(* IEC 61131-3 sources: thecodesysvibecoder/templates, 10 files *)

(* ---- FB_EtherCATMasterRestart.decl.st ---- *)
FUNCTION_BLOCK FB_EtherCATMasterRestart
VAR_INPUT
    xExecute : BOOL; // Rising edge starts a restart/reconfigure of the EtherCAT master connector.
    dwMasterModuleType : DWORD := DWORD#16#40; // IoStandard connector type CT_ETHERCAT_MASTER.
    dwMasterInstance : DWORD := 0; // EtherCAT master connector instance; normally 0 when there is one master.
END_VAR
VAR_OUTPUT
    xBusy : BOOL; // TRUE while IoMgrReconfigure is active.
    xDone : BOOL; // One-cycle pulse when the restart/reconfigure reports ASYNCSTATE_READY.
    xError : BOOL; // TRUE if the master connector cannot be found or reconfigure reports an error.
    xConnectorFound : BOOL; // TRUE when the EtherCAT master connector is found in the IoMgr connector list.
    dwMasterFlags : DWORD; // Raw IoConfigConnector.dwFlags of the master connector.
    udiConfigResult : UDINT; // Return code from IoMgrConfigGetConnectorList.
    udiReconfigureResult : UDINT; // Return code from IoMgrReconfigure.
    udiAsyncState : UDINT; // Async state: 0=pending, 1=active, 2=ready, 3=error, 4=timeout.
END_VAR
VAR
    pConnectorList : POINTER TO IoConfigConnector;
    pMasterConnector : POINTER TO IoConfigConnector;
    pActiveConnector : POINTER TO IoConfigConnector;
    diConnectorCount : DINT;
    xPrevExecute : BOOL; // Previous xExecute value for rising-edge detection.
    xStartRequest : BOOL; // Internal one-cycle request trigger.
    uiState : UINT; // 0=idle, 10=reconfigure active.
END_VAR

(* ---- FB_EtherCATOptionalSlaveManager.decl.st ---- *)
FUNCTION_BLOCK FB_EtherCATOptionalSlaveManager
VAR_INPUT
    xEnable : BOOL := TRUE; // FALSE leaves the EtherCAT master untouched by this FB.
    uiRequiredSlaves : UINT := 1; // Number of configured slaves that must be present; higher indexed slaves become optional.
    xApply : BOOL; // Rising edge reapplies optional flags and optionally restarts the master.
    xAutoApplyOnChange : BOOL := TRUE; // TRUE reapplies when uiRequiredSlaves changes.
    xRestartAfterApply : BOOL := TRUE; // TRUE pulses EtherCAT_Master.xRestart after optional flags are changed.
    xRestart : BOOL; // Manual rising edge pulses EtherCAT_Master.xRestart.
    xStepNonOperationalToOp : BOOL := TRUE; // TRUE tries INIT->PREOP->SAFEOP->OP for required slaves not yet operational.
    xStartConfigWithLessDevice : BOOL := TRUE; // Allows startup when optional configured slaves are not physically present.
    xAutoSetOperational : BOOL := TRUE; // Lets the master automatically retry optional/returning slaves.
    uiMaxSlavesToScan : UINT := 32; // Loop guard for the generated EtherCAT slave chain.
END_VAR
VAR_OUTPUT
    xDone : BOOL; // One-cycle pulse after optional flags were applied.
    xRestartPulse : BOOL; // TRUE for the cycle in which EtherCAT_Master.xRestart is pulsed.
    xConfigFinished : BOOL; // EtherCAT master reports that configuration download/startup is finished.
    xMasterError : BOOL; // EtherCAT master error output.
    xAnyNonOperational : BOOL; // TRUE when at least one scanned slave is not OP.
    uiConfiguredSlaves : UINT; // Number of slaves reached through EtherCAT_Master.FirstSlave/NextInstance.
    uiOptionalSlaves : UINT; // Number of scanned slaves above uiRequiredSlaves.
    uiOperationalSlaves : UINT; // Number of scanned slaves currently in OP.
    uiFirstNonOperationalIndex : UINT; // 1-based index of the first scanned slave not in OP; 0 when all are OP.
    eFirstNonOperationalState : ETC_SLAVE_STATE; // State of the first non-OP slave.
END_VAR
VAR
    pSlave : POINTER TO ETCSlave;
    uiIndex : UINT;
    xPrevApply : BOOL;
    xPrevRestart : BOOL;
    uiPrevRequiredSlaves : UINT := 65535;
    xApplyRequest : BOOL;
    xManualRestartRequest : BOOL;
    xDoRestart : BOOL;
    xOptional : BOOL;
END_VAR

(* ---- FB_IoConnectorRuntimeEnable.decl.st ---- *)
FUNCTION_BLOCK FB_IoConnectorRuntimeEnable
VAR_INPUT
    xEnable : BOOL := TRUE; // Requested runtime state for the selected I/O connector.
    xApply : BOOL; // Optional rising edge that applies the current request immediately.
    xAutoApplyOnChange : BOOL := TRUE; // TRUE applies automatically whenever xEnable changes.
    dwModuleType : DWORD := DWORD#16#41; // IoStandard module type; 16#41 is an EtherCAT slave connector in this project.
    dwInstance : DWORD := 1; // Connector instance: normally 0=first EtherCAT slave, 1=second, 2=third, etc.
    xUseCachedConnector : BOOL := TRUE; // Allows re-enable when a disabled connector is no longer returned by the active list.
END_VAR
VAR_OUTPUT
    xBusy : BOOL; // TRUE while IoMgrReconfigure is active.
    xDone : BOOL; // One-cycle pulse when reconfiguration reports ASYNCSTATE_READY.
    xError : BOOL; // TRUE if no usable connector exists or reconfiguration reports an error.
    xConnectorFound : BOOL; // TRUE when the connector is found in the current IoMgr connector list.
    xTargetAvailable : BOOL; // TRUE when either the current connector or a cached connector can be used.
    xUsingCachedConnector : BOOL; // TRUE when the FB is using the cached connector pointer for this cycle.
    xCurrentEnable : BOOL; // Current CF_ENABLE + CF_DEVICE_ENABLED flag state on the target connector.
    dwCurrentFlags : DWORD; // Raw IoConfigConnector.dwFlags of the target connector.
    udiConfigResult : UDINT; // Return code from IoMgrConfigGetConnectorList.
    udiReconfigureResult : UDINT; // Return code from IoMgrReconfigure.
    udiAsyncState : UDINT; // Async state: 0=pending, 1=active, 2=ready, 3=error, 4=timeout.
END_VAR
VAR
    pConnectorList : POINTER TO IoConfigConnector;
    pFoundConnector : POINTER TO IoConfigConnector;
    pTargetConnector : POINTER TO IoConfigConnector;
    pCachedConnector : POINTER TO IoConfigConnector;
    pActiveConnector : POINTER TO IoConfigConnector;
    diConnectorCount : DINT;
    xHaveCachedConnector : BOOL; // TRUE after the target connector was found at least once.
    xPrevApply : BOOL; // Previous xApply value for rising-edge detection.
    xPrevEnable : BOOL := TRUE; // Previous xEnable value for automatic change detection.
    xStartRequest : BOOL; // Internal one-cycle request trigger.
    uiState : UINT; // 0=idle, 10=reconfigure active.
END_VAR

(* ---- FB_MD5Hash.decl.st ---- *)
FUNCTION_BLOCK FB_MD5Hash
VAR_INPUT
    xExecute : BOOL; // Rising edge starts a new MD5 calculation.
    pData : POINTER TO BYTE; // Start address of the data to hash, normally ADR(stYourData).
    udiSize : UDINT; // Number of bytes to hash, normally SIZEOF(stYourData).
    abyExpectedDigest : ARRAY [0..15] OF BYTE; // Optional MD5 digest received from the other controller.
    xCompareExpected : BOOL := TRUE; // When TRUE, xMatch is updated when the local digest is done.
END_VAR
VAR_OUTPUT
    xDone : BOOL; // TRUE after a successful calculation; reset by the next xExecute rising edge.
    xBusy : BOOL; // TRUE while the CAA Memory MD5 block is calculating.
    xError : BOOL; // TRUE if a request is invalid, for example null pointer or zero byte length.
    xMatch : BOOL; // TRUE when the calculated digest equals abyExpectedDigest.
    abyDigest : ARRAY [0..15] OF BYTE; // Calculated 16-byte MD5 digest.
END_VAR
VAR
    fbMd5 : MEM.MD5; // CAA Memory MD5 function block.
    xExecuteOld : BOOL; // Previous xExecute state for rising-edge detection.
    xStart : BOOL; // One-cycle start pulse forwarded to MEM.MD5.
    i : INT; // Digest byte loop index.
END_VAR

(* ---- FB_S10eRuntimeEnable.decl.st ---- *)
FUNCTION_BLOCK FB_S10eRuntimeEnable
VAR_INPUT
    xEnableS10e1 : BOOL := TRUE; // Requested runtime state for the selected S10e EtherCAT slave.
    xApply : BOOL; // Optional rising edge that applies the current request immediately.
    xAutoApplyOnChange : BOOL := TRUE; // TRUE applies automatically whenever xEnableS10e1 changes.
    dwSlaveInstance : DWORD := 1; // Connector instance: normally 0=first S10e, 1=second, 2=third, etc.
    dwModuleType : DWORD := DWORD#16#41; // IoStandard module type; 16#41 is an EtherCAT slave connector in this project.
    xUseCachedConnector : BOOL := TRUE; // Allows re-enable when a disabled connector is no longer returned by the active list.
END_VAR
VAR_OUTPUT
    xBusy : BOOL; // TRUE while IoMgrReconfigure is active.
    xDone : BOOL; // One-cycle pulse when reconfiguration reports ASYNCSTATE_READY.
    xError : BOOL; // TRUE if no usable connector exists or reconfiguration reports an error.
    xConnectorFound : BOOL; // TRUE when the connector is found in the current IoMgr connector list.
    xTargetAvailable : BOOL; // TRUE when either the current connector or a cached connector can be used.
    xUsingCachedConnector : BOOL; // TRUE when the FB is using the cached connector pointer for this cycle.
    xCurrentEnable : BOOL; // Current CF_ENABLE + CF_DEVICE_ENABLED flag state on the target connector.
    dwCurrentFlags : DWORD; // Raw IoConfigConnector.dwFlags of the target connector.
    udiConfigResult : UDINT; // Return code from IoMgrConfigGetConnectorList.
    udiReconfigureResult : UDINT; // Return code from IoMgrReconfigure.
    udiAsyncState : UDINT; // Async state: 0=pending, 1=active, 2=ready, 3=error, 4=timeout.
END_VAR
VAR
    pConnectorList : POINTER TO IoConfigConnector;
    pFoundConnector : POINTER TO IoConfigConnector;
    pTargetConnector : POINTER TO IoConfigConnector;
    pCachedConnector : POINTER TO IoConfigConnector;
    pActiveConnector : POINTER TO IoConfigConnector;
    diConnectorCount : DINT;
    xHaveCachedConnector : BOOL; // TRUE after the target connector was found at least once.
    xPrevApply : BOOL; // Previous xApply value for rising-edge detection.
    xPrevEnableS10e1 : BOOL := TRUE; // Previous enable request for auto-apply change detection.
    xStartRequest : BOOL; // Internal one-cycle request trigger.
    uiState : UINT; // 0=idle, 10=reconfigure active.
END_VAR

(* ---- FB_EtherCATMasterRestart.impl.st ---- *)
// Restart/reconfigure the complete EtherCAT master connector.
// IoMgrReconfigure performs an asynchronous disable/enable/update-mapping
// sequence for the connector, which is the closest runtime "master restart"
// available through IoStandard.
xDone := FALSE;
xStartRequest := FALSE;

IF xExecute AND NOT xPrevExecute THEN
    xStartRequest := TRUE;
END_IF
xPrevExecute := xExecute;

udiConfigResult := IoMgrConfigGetConnectorList(
    ppConnectorList := ADR(pConnectorList),
    pnCount := ADR(diConnectorCount));

pMasterConnector := IoMgrConfigGetConnector(
    pConnectorList := pConnectorList,
    pnCount := ADR(diConnectorCount),
    dwModuleType := dwMasterModuleType,
    dwInstance := dwMasterInstance);

IF pMasterConnector <> 0 THEN
    xConnectorFound := TRUE;
    dwMasterFlags := pMasterConnector^.dwFlags;
ELSE
    xConnectorFound := FALSE;
    dwMasterFlags := DWORD#0;
END_IF

CASE uiState OF
    0:
        xBusy := FALSE;
        udiReconfigureResult := UDINT#0;

        IF xStartRequest THEN
            IF (udiConfigResult <> UDINT#0) OR NOT xConnectorFound THEN
                xError := TRUE;
            ELSE
                xError := FALSE;
                udiAsyncState := UDINT#16#FFFFFFFF;
                pActiveConnector := pMasterConnector;
                uiState := 10;
            END_IF
        END_IF

    10:
        xBusy := TRUE;
        IF pActiveConnector = 0 THEN
            xBusy := FALSE;
            xError := TRUE;
            uiState := 0;
        ELSE
            udiReconfigureResult := IoMgrReconfigure(
                pConnector := pActiveConnector,
                pudiState := ADR(udiAsyncState));

            dwMasterFlags := pActiveConnector^.dwFlags;

            IF udiReconfigureResult <> UDINT#0 THEN
                xBusy := FALSE;
                xError := TRUE;
                uiState := 0;
            ELSIF udiAsyncState = UDINT#2 THEN
                xBusy := FALSE;
                xDone := TRUE;
                xError := FALSE;
                uiState := 0;
            ELSIF (udiAsyncState = UDINT#3) OR (udiAsyncState = UDINT#4) THEN
                xBusy := FALSE;
                xError := TRUE;
                uiState := 0;
            END_IF
        END_IF

ELSE
    xBusy := FALSE;
    xError := TRUE;
    uiState := 0;
END_CASE

(* ---- FB_EtherCATOptionalSlaveManager.impl.st ---- *)
// Use the EtherCAT driver's optional-slave support instead of disabling
// IoStandard connectors. Disabled connectors can disappear from the runtime
// configuration and may not come back until a controller warm restart.
xDone := FALSE;
xRestartPulse := FALSE;
xApplyRequest := FALSE;
xManualRestartRequest := FALSE;

IF NOT xEnable THEN
    RETURN;
END_IF

IF xApply AND NOT xPrevApply THEN
    xApplyRequest := TRUE;
END_IF

IF xRestart AND NOT xPrevRestart THEN
    xManualRestartRequest := TRUE;
END_IF

IF xAutoApplyOnChange AND (uiRequiredSlaves <> uiPrevRequiredSlaves) THEN
    xApplyRequest := TRUE;
END_IF

xPrevApply := xApply;
xPrevRestart := xRestart;

// These properties must be set before or while the master starts.
EtherCAT_Master.StartConfigWithLessDevice := xStartConfigWithLessDevice;
EtherCAT_Master.AutoSetOperational := xAutoSetOperational;

IF xApplyRequest THEN
    pSlave := EtherCAT_Master.FirstSlave;
    uiIndex := 1;

    WHILE (pSlave <> 0) AND (uiIndex <= uiMaxSlavesToScan) DO
        // Slaves after uiRequiredSlaves remain in the configuration but are optional.
        xOptional := uiIndex > uiRequiredSlaves;
        pSlave^.SetOptional(xOptional);

        pSlave := pSlave^.NextInstance;
        uiIndex := uiIndex + 1;
    END_WHILE

    uiPrevRequiredSlaves := uiRequiredSlaves;
    xDone := TRUE;
END_IF

xDoRestart := xManualRestartRequest OR (xApplyRequest AND xRestartAfterApply);
EtherCAT_Master.xRestart := xDoRestart;
xRestartPulse := xDoRestart;

// The generated master instance must be called for xRestart and status updates.
EtherCAT_Master();

xConfigFinished := EtherCAT_Master.xConfigFinished;
xMasterError := EtherCAT_Master.xError;

uiConfiguredSlaves := 0;
uiOptionalSlaves := 0;
uiOperationalSlaves := 0;
uiFirstNonOperationalIndex := 0;
xAnyNonOperational := FALSE;
eFirstNonOperationalState := ETC_SLAVE_STATE.ETC_SLAVE_BOOT;

pSlave := EtherCAT_Master.FirstSlave;
uiIndex := 1;

WHILE (pSlave <> 0) AND (uiIndex <= uiMaxSlavesToScan) DO
    pSlave^();
    uiConfiguredSlaves := uiConfiguredSlaves + 1;

    xOptional := uiIndex > uiRequiredSlaves;
    IF xOptional THEN
        uiOptionalSlaves := uiOptionalSlaves + 1;
    END_IF

    IF pSlave^.wState = ETC_SLAVE_STATE.ETC_SLAVE_OPERATIONAL THEN
        uiOperationalSlaves := uiOperationalSlaves + 1;
    ELSE
        xAnyNonOperational := TRUE;
        IF uiFirstNonOperationalIndex = 0 THEN
            uiFirstNonOperationalIndex := uiIndex;
            eFirstNonOperationalState := pSlave^.wState;
        END_IF

        // Required slaves are actively stepped toward OP. Optional slaves are
        // handled by AutoSetOperational when they are connected again.
        IF xStepNonOperationalToOp AND xConfigFinished AND NOT xOptional THEN
            CASE pSlave^.wState OF
                ETC_SLAVE_STATE.ETC_SLAVE_INIT:
                    pSlave^.SetOpMode(ETC_SLAVE_STATE.ETC_SLAVE_PREOPERATIONAL);
                ETC_SLAVE_STATE.ETC_SLAVE_PREOPERATIONAL:
                    pSlave^.SetOpMode(ETC_SLAVE_STATE.ETC_SLAVE_SAVEOPERATIONAL);
                ETC_SLAVE_STATE.ETC_SLAVE_SAVEOPERATIONAL:
                    pSlave^.SetOpMode(ETC_SLAVE_STATE.ETC_SLAVE_OPERATIONAL);
            END_CASE
        END_IF
    END_IF

    pSlave := pSlave^.NextInstance;
    uiIndex := uiIndex + 1;
END_WHILE

(* ---- FB_IoConnectorRuntimeEnable.impl.st ---- *)
// Generic low-level runtime enable/disable for an IoStandard connector.
// For S10e EtherCAT slaves in this project, use dwModuleType 16#41 and select
// the unit by dwInstance. The CODESYS object name is not needed at runtime.
xDone := FALSE;
xStartRequest := FALSE;
xUsingCachedConnector := FALSE;

IF xApply AND NOT xPrevApply THEN
    xStartRequest := TRUE;
END_IF

IF xAutoApplyOnChange AND (xEnable <> xPrevEnable) THEN
    xStartRequest := TRUE;
END_IF

xPrevApply := xApply;
xPrevEnable := xEnable;

udiConfigResult := IoMgrConfigGetConnectorList(
    ppConnectorList := ADR(pConnectorList),
    pnCount := ADR(diConnectorCount));

pFoundConnector := IoMgrConfigGetConnector(
    pConnectorList := pConnectorList,
    pnCount := ADR(diConnectorCount),
    dwModuleType := dwModuleType,
    dwInstance := dwInstance);

IF pFoundConnector <> 0 THEN
    xConnectorFound := TRUE;
    pTargetConnector := pFoundConnector;
    pCachedConnector := pFoundConnector;
    xHaveCachedConnector := TRUE;
ELSE
    xConnectorFound := FALSE;

    IF xUseCachedConnector AND xHaveCachedConnector THEN
        pTargetConnector := pCachedConnector;
        xUsingCachedConnector := TRUE;
    ELSE
        pTargetConnector := 0;
    END_IF
END_IF

IF pTargetConnector <> 0 THEN
    xTargetAvailable := TRUE;
    dwCurrentFlags := pTargetConnector^.dwFlags;
    xCurrentEnable := (pTargetConnector^.dwFlags AND DWORD#16#5) = DWORD#16#5;
ELSE
    xTargetAvailable := FALSE;
    dwCurrentFlags := DWORD#0;
    xCurrentEnable := FALSE;
END_IF

CASE uiState OF
    0:
        xBusy := FALSE;
        udiReconfigureResult := UDINT#0;

        IF xStartRequest THEN
            IF (udiConfigResult <> UDINT#0) OR NOT xTargetAvailable THEN
                xError := TRUE;
            ELSE
                xError := FALSE;
                udiAsyncState := UDINT#16#FFFFFFFF;

                IF xEnable THEN
                    pTargetConnector^.dwFlags := pTargetConnector^.dwFlags OR DWORD#16#5;
                ELSE
                    pTargetConnector^.dwFlags := pTargetConnector^.dwFlags AND DWORD#16#FFFFFFFA;
                END_IF

                pActiveConnector := pTargetConnector;
                pCachedConnector := pTargetConnector;
                xHaveCachedConnector := TRUE;
                dwCurrentFlags := pTargetConnector^.dwFlags;
                xCurrentEnable := (pTargetConnector^.dwFlags AND DWORD#16#5) = DWORD#16#5;
                uiState := 10;
            END_IF
        END_IF

    10:
        xBusy := TRUE;
        IF pActiveConnector = 0 THEN
            xBusy := FALSE;
            xError := TRUE;
            uiState := 0;
        ELSE
            udiReconfigureResult := IoMgrReconfigure(
                pConnector := pActiveConnector,
                pudiState := ADR(udiAsyncState));

            dwCurrentFlags := pActiveConnector^.dwFlags;
            xCurrentEnable := (pActiveConnector^.dwFlags AND DWORD#16#5) = DWORD#16#5;

            IF udiReconfigureResult <> UDINT#0 THEN
                xBusy := FALSE;
                xError := TRUE;
                uiState := 0;
            ELSIF udiAsyncState = UDINT#2 THEN
                xBusy := FALSE;
                xDone := TRUE;
                xError := FALSE;
                uiState := 0;
            ELSIF (udiAsyncState = UDINT#3) OR (udiAsyncState = UDINT#4) THEN
                xBusy := FALSE;
                xError := TRUE;
                uiState := 0;
            END_IF
        END_IF

ELSE
    xBusy := FALSE;
    xError := TRUE;
    uiState := 0;
END_CASE

(* ---- FB_MD5Hash.impl.st ---- *)
// Create a one-cycle start pulse. The wrapped MEM.MD5 block starts on a rising edge.
xStart := xExecute AND NOT xExecuteOld;
xExecuteOld := xExecute;

IF xStart THEN
    xDone := FALSE;
    xError := FALSE;
    xMatch := FALSE;
END_IF

// Reject invalid requests before forwarding the start pulse to the library block.
IF xStart AND ((pData = 0) OR (udiSize = 0)) THEN
    xError := TRUE;
END_IF

fbMd5(
    xExecute := xStart AND NOT xError,
    pMemoryBlock := pData,
    udiNumberOfBytes := udiSize
);

xBusy := fbMd5.xBusy;

IF fbMd5.xDone THEN
    // Copy the library digest to stable wrapper outputs.
    FOR i := 0 TO 15 DO
        abyDigest[i] := fbMd5.abyDigest[i];
    END_FOR

    xDone := TRUE;

    // Compare byte-for-byte with the digest supplied by the communication peer.
    IF xCompareExpected THEN
        xMatch := TRUE;
        FOR i := 0 TO 15 DO
            IF abyDigest[i] <> abyExpectedDigest[i] THEN
                xMatch := FALSE;
            END_IF
        END_FOR
    END_IF
END_IF

(* ---- FB_S10eRuntimeEnable.impl.st ---- *)
// Low-level runtime enable/disable for an S10e EtherCAT slave connector.
// The unit is selected by connector instance, so the CODESYS object name is
// not needed at runtime. A cached connector pointer is kept because a disabled
// connector may disappear from the active connector list before it is enabled.
xDone := FALSE;
xStartRequest := FALSE;
xUsingCachedConnector := FALSE;

IF xApply AND NOT xPrevApply THEN
    xStartRequest := TRUE;
END_IF

IF xAutoApplyOnChange AND (xEnableS10e1 <> xPrevEnableS10e1) THEN
    xStartRequest := TRUE;
END_IF

xPrevApply := xApply;
xPrevEnableS10e1 := xEnableS10e1;

udiConfigResult := IoMgrConfigGetConnectorList(
    ppConnectorList := ADR(pConnectorList),
    pnCount := ADR(diConnectorCount));

pFoundConnector := IoMgrConfigGetConnector(
    pConnectorList := pConnectorList,
    pnCount := ADR(diConnectorCount),
    dwModuleType := dwModuleType,
    dwInstance := dwSlaveInstance);

IF pFoundConnector <> 0 THEN
    xConnectorFound := TRUE;
    pTargetConnector := pFoundConnector;
    pCachedConnector := pFoundConnector;
    xHaveCachedConnector := TRUE;
ELSE
    xConnectorFound := FALSE;

    IF xUseCachedConnector AND xHaveCachedConnector THEN
        pTargetConnector := pCachedConnector;
        xUsingCachedConnector := TRUE;
    ELSE
        pTargetConnector := 0;
    END_IF
END_IF

IF pTargetConnector <> 0 THEN
    xTargetAvailable := TRUE;
    dwCurrentFlags := pTargetConnector^.dwFlags;
    xCurrentEnable := (pTargetConnector^.dwFlags AND DWORD#16#5) = DWORD#16#5;
ELSE
    xTargetAvailable := FALSE;
    dwCurrentFlags := DWORD#0;
    xCurrentEnable := FALSE;
END_IF

CASE uiState OF
    0:
        xBusy := FALSE;
        udiReconfigureResult := UDINT#0;

        IF xStartRequest THEN
            IF (udiConfigResult <> UDINT#0) OR NOT xTargetAvailable THEN
                xError := TRUE;
            ELSE
                xError := FALSE;
                udiAsyncState := UDINT#16#FFFFFFFF;

                IF xEnableS10e1 THEN
                    pTargetConnector^.dwFlags := pTargetConnector^.dwFlags OR DWORD#16#5;
                ELSE
                    pTargetConnector^.dwFlags := pTargetConnector^.dwFlags AND DWORD#16#FFFFFFFA;
                END_IF

                pActiveConnector := pTargetConnector;
                pCachedConnector := pTargetConnector;
                xHaveCachedConnector := TRUE;
                dwCurrentFlags := pTargetConnector^.dwFlags;
                xCurrentEnable := (pTargetConnector^.dwFlags AND DWORD#16#5) = DWORD#16#5;
                uiState := 10;
            END_IF
        END_IF

    10:
        xBusy := TRUE;
        IF pActiveConnector = 0 THEN
            xBusy := FALSE;
            xError := TRUE;
            uiState := 0;
        ELSE
            udiReconfigureResult := IoMgrReconfigure(
                pConnector := pActiveConnector,
                pudiState := ADR(udiAsyncState));

            dwCurrentFlags := pActiveConnector^.dwFlags;
            xCurrentEnable := (pActiveConnector^.dwFlags AND DWORD#16#5) = DWORD#16#5;

            IF udiReconfigureResult <> UDINT#0 THEN
                xBusy := FALSE;
                xError := TRUE;
                uiState := 0;
            ELSIF udiAsyncState = UDINT#2 THEN
                xBusy := FALSE;
                xDone := TRUE;
                xError := FALSE;
                uiState := 0;
            ELSIF (udiAsyncState = UDINT#3) OR (udiAsyncState = UDINT#4) THEN
                xBusy := FALSE;
                xError := TRUE;
                uiState := 0;
            END_IF
        END_IF

ELSE
    xBusy := FALSE;
    xError := TRUE;
    uiState := 0;
END_CASE
